TYPE RecipeAxisLinear2Pos_t :
STRUCT
    rPosGS    : REAL;
    rPosAS    : REAL;
    rVeloToAS : REAL;
    rVeloToGS : REAL;
    rAccel    : REAL;
    rDecel    : REAL;
    rJerk     : REAL;
END_STRUCT
END_TYPE

(* stored: Version 1.1.0.1, ProductVersion 3.1.4024.6
   DUT RecipeAxisLinear2Pos_t: Id {d2ed1bb6-1652-4dc7-ab10-3b29c78e467b} *)
